Fanuc KAREL source: CREATE_VAR.kl

PROGRAM T
%NOLOCKGROUP
VAR
 v0 : STRING[40]
 v1 : STRING[40]
 v2 : STRING[40]
 v3 : STRING[40]
 v4 : INTEGER
 v5 : INTEGER
 v6 : INTEGER
 v7 : INTEGER
 v8 : INTEGER
BEGIN
 CREATE_VAR(v0, v1, v2, v3, v4, v5, v6, v7, v8)
END T
